{attribute 'qualified_only'}
{attribute 'strict'}
TYPE nHP_Axis_AdjustmentModes :
(
	None := 0,
	FitByABS := 1,
	FitByDRM := 2,
	FitByForfce := 3
);
END_TYPE

(* stored: Version 1.1.0.1, ProductVersion 3.1.4024.15
   EnumerationTextList nHP_Axis_AdjustmentModes: Id {db58ba8b-d863-490c-b09e-46c9b83522b9} *)
